SUBAPPLICATION Uebung_082 (* Beispiel für E_CTUD *)
  (* Standard: 61499-2; Description: Beispiel für E_CTD Aufwärts zählen UAO Curriculum Module 3 - The IEC 61499 Standard, Seite 94 *)
  (* Version 1.0, 2023-10-23, franz *)
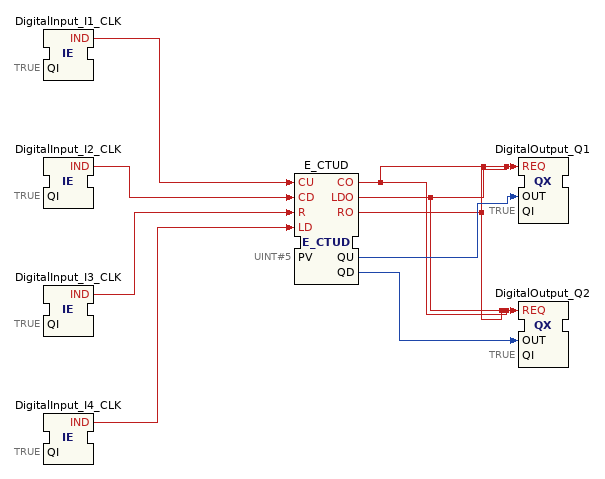
  FBS
    DigitalOutput_Q1 : QX(QI := TRUE);
    DigitalInput_I1_CLK : IE(QI := TRUE);
    E_CTUD : E_CTUD(PV := UINT#5);
    DigitalInput_I2_CLK : IE(QI := TRUE);
    DigitalInput_I3_CLK : IE(QI := TRUE);
    DigitalInput_I4_CLK : IE(QI := TRUE);
    DigitalOutput_Q2 : QX(QI := TRUE);
  END_FBS
  EVENT_CONNECTIONS
    DigitalInput_I1_CLK.IND TO E_CTUD.CU;
    E_CTUD.CO TO DigitalOutput_Q1.REQ;
    E_CTUD.LDO TO DigitalOutput_Q1.REQ;
    DigitalInput_I2_CLK.IND TO E_CTUD.CD;
    E_CTUD.RO TO DigitalOutput_Q1.REQ;
    DigitalInput_I3_CLK.IND TO E_CTUD.R;
    DigitalInput_I4_CLK.IND TO E_CTUD.LD;
    E_CTUD.LDO TO DigitalOutput_Q2.REQ;
    E_CTUD.CO TO DigitalOutput_Q2.REQ;
    E_CTUD.RO TO DigitalOutput_Q2.REQ;
  END_CONNECTIONS
  DATA_CONNECTIONS
    E_CTUD.QU TO DigitalOutput_Q1.OUT;
    E_CTUD.QD TO DigitalOutput_Q2.OUT;
  END_CONNECTIONS
END_SUBAPPLICATION
